(* PLC project PLC, Beckhoff Automation GmbH TwinCAT PLC Control 3.5.10.30 *)
(* stored: creationDateTime 2019-05-17T10:29:43.5973623, modificationDateTime 2019-05-17T10:29:43.6023611 *)

// Treats supplied array (of any type) as First-in First-out queue.
// Usage: fbFifoQueue(ptrArrData:=ADR(queue_array), Length:=[array length], Ring:=[true/false]);
FUNCTION_BLOCK FB_FifoQueue
VAR_INPUT
	ptrArrData 	: POINTER TO DWORD; // Queue Data Array
	Length 		: DINT;				// Length of Queue
	Ring		: BOOL;				// Queue acts as a Ring Buffer (oldest data is overwritten when queue is full)
END_VAR
VAR_OUTPUT
END_VAR
VAR
	// pointer to enqueue (head) element
	_ptrEnqueue 	: POINTER TO DWORD;
	// pointer to dequeue (tail) element
	_ptrDequeue	: POINTER TO DWORD;
	
	// queue/dequeue indices
	_idxEnqueue	: DINT;
	_idxDequeue	: DINT;
	
	// element count
	_count 		: DINT;
	// buffer full
	_full 		: BOOL := FALSE;
	// buffer empty
	_empty 		: BOOL := TRUE;
	// element size
	_sizeof : DINT;
END_VAR

            
          

METHOD Clear
VAR_INPUT
END_VAR
                  // throw new NotImplementedException
                
END_METHOD

// Remove/Retrieve and item from the Queue. Returns a pointer to the retrieved item.
// Usage: MEMCPY(ADR(destination), fbFifoQueue.Dequeue(), SIZEOF(destination));
METHOD Dequeue : POINTER TO DWORD
                  // reset full
_full := FALSE;

// queue has (valid) elements
IF _count > 0 AND _sizeof > 0 THEN
	
	// assign return value ptr
	Dequeue := _ptrDequeue;
	
	// increment pop ptr
	_idxDequeue := (_idxDequeue + 1) MOD Length;
	_ptrDequeue := ptrArrData + DINT_TO_DWORD(_sizeof * _idxDequeue);
	
	// decrement element count
	_count := _count - 1;
END_IF

// set empty
IF _count = 0 THEN
	_empty := TRUE;
END_IF
                
END_METHOD

// Add an item to the Queue.
// Usage: fbFifoQueue.Enqueue(item);
METHOD Enqueue
VAR_INPUT
	Val : ANY;	// Queued Item
END_VAR
                  // reset empty
_empty := FALSE;

// if first call to enqueue
IF _ptrEnqueue = 0 THEN
	
	// initialize pointers
	_ptrEnqueue := ptrArrData;
	_ptrDequeue := _ptrEnqueue;
	
	// get element size
	_sizeof := Val.diSize;
END_IF

// only overwrite data if in Ring buffer mode
IF (NOT _full) OR (_full AND Ring) THEN
	
	IF (_full AND Ring) THEN
		// increment dequeue ptr
		_idxDequeue := (_idxDequeue + 1) MOD Length;
		_ptrDequeue := ptrArrData + DINT_TO_DWORD(_sizeof * _idxDequeue);
	END_IF
	
	// load value into buffer
	MEMCPY(_ptrEnqueue, Val.pValue, DINT_TO_UDINT(_sizeof));

	// increment enqueue ptr
	_idxEnqueue := (_idxEnqueue + 1) MOD Length;
	_ptrEnqueue := ptrArrData + DINT_TO_DWORD(_sizeof * _idxEnqueue);
	
	// increment element count
	IF NOT _full THEN 
		_count := _count + 1; 
	END_IF
END_IF

// buffer full
IF _count = Length THEN
	_full := TRUE;
END_IF
                
END_METHOD

PROPERTY Count : DINT
GET
VAR
END_VAR
                    Count := _count;
                  
END_GET
END_PROPERTY

PROPERTY IsEmpty : BOOL
GET
VAR
END_VAR
                    IsEmpty := _empty;
                  
END_GET
END_PROPERTY

PROPERTY IsFull : BOOL
GET
VAR
END_VAR
                    IsFull := _full;
                  
END_GET
END_PROPERTY
END_FUNCTION_BLOCK
